END_VAR
VAR
	tCheckingFVP:							TON;//Таймер проеврки ФВН
	tStopTMP:								TON;//Таймер отановки УВП
	tOpenBAV3:								TON;
	iVacuumCameraProcessStage:				INT;//Стадия работывакуумной камеры   
	iCallbackStage:							INT;//Стадия с которой произошел переход в ошибку
	iVacuumCameraLastProcessStage:			INT;//Предыдущая стадия процесса вакуумной камеры
	iVacuumCameraNextProcessStage:			INT;//Следующая стадия процесса вакуумной камеры
	wStatus:								WORD;//Cтатус работы
	xVacuumCameraDevicesAutomode:			BOOL;//Все устрйоства вакуумной камеры в автоматическом режиме
	xLockCommand:							BOOL;//Сигнал о блокировки ввода новой комманды
	xStartFVPCheckinTimerFlag:				BOOL;//Флаг запуска таймера проверки насоса.
	xOpenBAV3timerFlag:						BOOL;
	xStopTMPTimerFlag:						BOOL;
END_VAR

VacuumCameraSetting.tStopTMPtime:=UDINT_TO_TIME((UINT_TO_UDINT(VacuumCameraSetting.uiStopTMPTimeSP)*1000));
VacuumCameraSetting.tOpenBAV3time:=UDINT_TO_TIME((UINT_TO_UDINT(VacuumCameraSetting.uiOpenBAV3TimeSP)*1000));
VacuumCameraSetting.uiStopTMPTimeLeft:=VacuumCameraSetting.uiStopTMPTimeLeft/1000;

tCheckingFVP.IN:=xStartFVPCheckinTimerFlag;
tCheckingFVP.PT:=T#60S;
tCheckingFVP();

tStopTMP.IN:=xStopTMPTimerFlag; 
tStopTMP.PT:=VacuumCameraSetting.tStopTMPtime;
VacuumCameraSetting.tStopTMPTimeLeft:=tStopTMP.ET;
tStopTMP();

tOpenBAV3.IN:=xOpenBAV3timerFlag;
tOpenBAV3.PT:=VacuumCameraSetting.tOpenBAV3time;
tOpenBAV3();


IF ClosedCameraSensore.xValue THEN
	VacuumCamera.xClosed:=TRUE;
ELSE
	VacuumCamera.xClosed:=FALSE;
END_IF

xVacuumCameraDevicesAutomode:=isVacuumCameraDeviceAutoMode;


CASE iVacuumCameraProcessStage OF
	

	VACUUM_CAMERA_PROCESS_STAGE.WAIT:	
	
		IF NOT xLockCommand  THEN
			OperatorCommandHandler();
		ELSE
			CancelOperatorCommand();
		END_IF
		IF xStopAnyProcessCommandFromOperator THEN
			iVacuumCameraNextProcessStage:=VACUUM_CAMERA_PROCESS_STAGE.STOP_ANY_PROCESS;
			xStopAnyProcessCommandFromOperator:=FALSE;
			Status:=VacuumCameraStatusList.STOP_ANY_PROCESS_SIGNAL_FROM_OPERATOR;
		END_IF
		IF NOT isVacuumCameraDeviceAutoMode AND xLockCommand THEN
			Status:=VacuumCameraStatusList.SYSTEM_HAS_ERROR;
			xError:=TRUE;
			wError:=VacuumCameraErrorsList.ALL_DEVICES_DONT_HAVE_AUTOMODE;
		END_IF
		IF xError THEN
			Status:=VacuumCameraStatusList.SYSTEM_HAS_ERROR;
			iVacuumCameraNextProcessStage:=VACUUM_CAMERA_PROCESS_STAGE.ERROR;
		END_IF
		iVacuumCameraProcessStage:=iVacuumCameraNextProcessStage;
		
	
	
	
	VACUUM_CAMERA_PROCESS_STAGE.START_VACUUM_PROCESS:
		iVacuumCameraLastProcessStage:=iVacuumCameraProcessStage;
		iCallBackStage:=iVacuumCameraProcessStage;
		Status:=startVacuumProcess();
		iVacuumCameraProcessStage:=VACUUM_CAMERA_PROCESS_STAGE.WAIT;
		
	VACUUM_CAMERA_PROCESS_STAGE.START_VACUUM_PROCESS_CHECK_FVP_SELECT:
		iVacuumCameraLastProcessStage:=iVacuumCameraProcessStage;
		iCallBackStage:=iVacuumCameraProcessStage;
		Status:=CheckFVPSelect();
		iVacuumCameraProcessStage:=VACUUM_CAMERA_PROCESS_STAGE.WAIT;
		
	VACUUM_CAMERA_PROCESS_STAGE.START_VACUUM_PROCESS_CHECKING_FVP:
		iVacuumCameraLastProcessStage:=iVacuumCameraProcessStage;
		iCallbackStage:=iVacuumCameraProcessStage;
		Status:=CheckingFVP();
		iVacuumCameraProcessStage:=VACUUM_CAMERA_PROCESS_STAGE.WAIT;
		
		
	VACUUM_CAMERA_PROCESS_STAGE.START_VACUUM_PROCESS_FORVACUUMING_PROCESS:
		iVacuumCameraLastProcessStage:=iVacuumCameraProcessStage;
		iCallbackStage:=iVacuumCameraProcessStage;
		Status:=forvacuumingProcess();
		iVacuumCameraProcessStage:=VACUUM_CAMERA_PROCESS_STAGE.WAIT;
		
	VACUUM_CAMERA_PROCESS_STAGE.START_VACUUM_PROCESS_TMP_FORVACUUMING_PROCESS:
		iVacuumCameraLastProcessStage:=iVacuumCameraProcessStage;
		iCallbackStage:=iVacuumCameraProcessStage;
		Status:=forvacuumingWithTMPValve();
		iVacuumCameraProcessStage:=VACUUM_CAMERA_PROCESS_STAGE.WAIT;
		
	VACUUM_CAMERA_PROCESS_STAGE.START_VACUUM_PROCESS_TMP_START:
		iVacuumCameraLastProcessStage:=iVacuumCameraProcessStage;
		iCallbackStage:=iVacuumCameraProcessStage;
		Status:=startTMP();
		iVacuumCameraProcessStage:=VACUUM_CAMERA_PROCESS_STAGE.WAIT;
	
	VACUUM_CAMERA_PROCESS_STAGE.START_VACUUM_PROCESS_COMPLETE_WAIT:
		iVacuumCameraLastProcessStage:=iVacuumCameraProcessStage;
		iCallbackStage:=iVacuumCameraProcessStage;
		Status:=waitVacuumingProcess();
		iVacuumCameraProcessStage:=VACUUM_CAMERA_PROCESS_STAGE.WAIT;
	
	
	VACUUM_CAMERA_PROCESS_STAGE.START_DEVACUUM_PROCESS:
		iVacuumCameraLastProcessStage:=iVacuumCameraProcessStage;
		iCallbackStage:=iVacuumCameraProcessStage;
		Status:=startDevacuumProcess();
		iVacuumCameraProcessStage:=VACUUM_CAMERA_PROCESS_STAGE.WAIT;
		
		
	VACUUM_CAMERA_PROCESS_STAGE.START_DEVACUUM_STOP_TMP:
		iVacuumCameraLastProcessStage:=iVacuumCameraProcessStage;
		iCallbackStage:=iVacuumCameraProcessStage;
		Status:=stopTMP();
		iVacuumCameraProcessStage:=VACUUM_CAMERA_PROCESS_STAGE.WAIT;

		
		
	VACUUM_CAMERA_PROCESS_STAGE.START_DEVACUUM_STOP_FVP:
		iVacuumCameraLastProcessStage:=iVacuumCameraProcessStage;
		iCallbackStage:=iVacuumCameraProcessStage;	
		Status:=stopFVP();
		iVacuumCameraProcessStage:=VACUUM_CAMERA_PROCESS_STAGE.WAIT;
		
	VACUUM_CAMERA_PROCESS_STAGE.START_DEVACUUM_OPEN_CAM:
		iVacuumCameraLastProcessStage:=iVacuumCameraProcessStage;
		iCallbackStage:=iVacuumCameraProcessStage;	
		Status:=devcuumProcessOpenCam();
		iVacuumCameraProcessStage:=VACUUM_CAMERA_PROCESS_STAGE.WAIT;
	
		
	VACUUM_CAMERA_PROCESS_STAGE.STOP_VACUUM_PROCESS:
		iVacuumCameraLastProcessStage:=iVacuumCameraProcessStage;
		iCallbackStage:=iVacuumCameraProcessStage;
		Status:=stopVacuumProcess();
		iVacuumCameraProcessStage:=VACUUM_CAMERA_PROCESS_STAGE.WAIT;
	
	VACUUM_CAMERA_PROCESS_STAGE.STOP_ANY_PROCESS:
		iVacuumCameraLastProcessStage:=iVacuumCameraProcessStage;
		iCallbackStage:=iVacuumCameraProcessStage;
		Status:=operatorStopAnyProcess();
		iVacuumCameraProcessStage:=VACUUM_CAMERA_PROCESS_STAGE.WAIT;
		
		
	VACUUM_CAMERA_PROCESS_STAGE.ERROR:
	
		ErrorHandle();
	
		
END_CASE

VacuumCamera.VacuumCameraProcessStage:=iVacuumCameraProcessStage;

ACTION StartDevacuumProcessCommand:
xStartDevacuumProcessOperatorCommand:=FALSE;
	IF isVacuumCameraDeviceAutoMode THEN
		iVacuumCameraNextProcessStage:=VACUUM_CAMERA_PROCESS_STAGE.START_DEVACUUM_PROCESS;
		xLockCommand:=TRUE;
		wError:=VacuumCameraErrorsList.NO_ERROR;
		RETURN;
	ELSE
		xError:=true;
		wError:=VacuumCameraErrorsList.ALL_DEVICES_DONT_HAVE_AUTOMODE;
		iVacuumCameraNextProcessStage:= VACUUM_CAMERA_PROCESS_STAGE.ERROR;
	END_IF
END_ACTION

ACTION StartVacuumProcessCommand:
	xStartVacuumProcessOperatorCommand:=FALSE;
	IF isVacuumCameraDeviceAutoMode THEN
		iVacuumCameraNextProcessStage:= VACUUM_CAMERA_PROCESS_STAGE.START_VACUUM_PROCESS;
		xLockCommand:=TRUE;
		wError:=VacuumCameraErrorsList.NO_ERROR;
		RETURN;
	END_IF
	IF NOT isVacuumCameraDeviceAutoMode THEN
		xError:=TRUE;
		wError:=VacuumCameraErrorsList.ALL_DEVICES_DONT_HAVE_AUTOMODE;
		iVacuumCameraNextProcessStage:= VACUUM_CAMERA_PROCESS_STAGE.ERROR;
	END_IF
	IF NOT VacuumCamera.xClosed THEN
		xError:=TRUE;
		wError:=VacuumCameraErrorsList.VACUUM_CAMERA_OPEN;
		iVacuumCameraNextProcessStage:= VACUUM_CAMERA_PROCESS_STAGE.ERROR;
	END_IF
END_ACTION

ACTION StopVacuumProcessCommand:
xStartVacuumProcessOperatorCommand:=FALSE;
IF isVacuumCameraDeviceAutoMode THEN
	iVacuumCameraNextProcessStage:=VACUUM_CAMERA_PROCESS_STAGE.STOP_VACUUM_PROCESS;
	xLockCommand:=TRUE;
	TMPBreakingValve.xAutoCommand:=FALSE;
	wError:=VacuumCameraErrorsList.NO_ERROR;
	RETURN;
ELSE
	xError:=TRUE;
	wError:=VacuumCameraErrorsList.ALL_DEVICES_DONT_HAVE_AUTOMODE;
	iVacuumCameraNextProcessStage:= VACUUM_CAMERA_PROCESS_STAGE.ERROR;
	
END_IF
END_ACTION

METHOD PROTECTED CancelOperatorCommand
VAR_INPUT
END_VAR
xStartVacuumProcessOperatorCommand:=FALSE;
xStartDevacuumProcessOperatorCommand:=FALSE;
xStopVacuumProcesOoperatorCommand:=FALSE;
END_METHOD

METHOD PROTECTED CheckFVPSelect : WORD
VAR_INPUT
END_VAR
IF NOT FVP.xStart THEN
			FVP.xAutoCommand:=TRUE;
			CheckFVPSelect:=VacuumCameraStatusList.CHECK_FVP_START_FVP;
END_IF
IF VacuumCamera.xFVPChecked THEN
			iVacuumCameraNextProcessStage:=VACUUM_CAMERA_PROCESS_STAGE.START_VACUUM_PROCESS_FORVACUUMING_PROCESS;
			CheckFVPSelect:=VacuumCameraStatusList.FVP_CHECK_COMPLETED;
ELSE
			iVacuumCameraNextProcessStage:=VACUUM_CAMERA_PROCESS_STAGE.START_VACUUM_PROCESS_CHECKING_FVP;
			xStartFVPCheckinTimerFlag:=TRUE;
END_IF
END_METHOD

METHOD PROTECTED CheckingFVP : WORD
VAR_INPUT
END_VAR
CheckingFVP:=VacuumCameraStatusList.CHECK_FVP_START_TIMER;		
IF tCheckingFVP.Q THEN
			IF FVPPressure.rPressure <= VacuumCameraSetting.rForvacPresureToCheckFVP THEN
				CheckingFVP:=VacuumCameraStatusList.CHECK_FVP_COMPLETE;
				VacuumCamera.xFVPChecked:=TRUE;
				iVacuumCameraNextProcessStage:=VACUUM_CAMERA_PROCESS_STAGE.START_VACUUM_PROCESS_FORVACUUMING_PROCESS;
			ELSE
				CheckingFVP:=VacuumCameraStatusList.CHECK_FVP_FAILED;
				iVacuumCameraNextProcessStage:=VACUUM_CAMERA_PROCESS_STAGE.ERROR;
				wError:=VacuumCameraErrorsList.FVP_CHECK_FAIL;
				xError:=TRUE;
			END_IF
	xStartFVPCheckinTimerFlag:=FALSE;
END_IF
END_METHOD

METHOD PROTECTED CloseAllvalves
VAR_INPUT
END_VAR
IF BAV1.xOpened THEN
	BAV1.xAutoCommand:=FALSE;
END_IF
IF BAV2.xOpened THEN
	BAV2.xAutoCommand:=FALSE;
END_IF
IF BAV3.xOpened THEN
	BAV3.xAutoCommand:=FALSE;
END_IF
IF TMPBreakingValve.xOpened THEN
	TMPBreakingValve.xAutoCommand:=FALSE;
END_IF
END_METHOD

METHOD PROTECTED devcuumProcessOpenCam : WORD
VAR_INPUT
END_VAR
IF BAV3.xClosed THEN
	BAV3.xAutoCommand:=TRUE;
	xOpenBAV3timerFlag:= TRUE;
	devcuumProcessOpenCam:=VacuumCameraStatusList.BAV3OPENED;
END_IF
IF tOpenBAV3.Q THEN
	xOpenBAV3timerFlag:=FALSE;
	BAV3.xAutoCommand:=FALSE;
	xLockCommand:=FALSE;
	devcuumProcessOpenCam:=VacuumCameraStatusList.STOP_SYSTEM_COMPLITE;
	iVacuumCameraNextProcessStage:= VACUUM_CAMERA_PROCESS_STAGE.WAIT;
END_IF
END_METHOD

METHOD PRIVATE ErrorHandle : WORD
VAR_INPUT
END_VAR
IF xProcessResumeCommand THEN
	xProcessResumeCommand:=FALSE;
	iVacuumCameraNextProcessStage:=iCallbackStage;
	iVacuumCameraProcessStage:=VACUUM_CAMERA_PROCESS_STAGE.WAIT;
	xError:=FALSE;
	wError:=VacuumCameraErrorsList.NO_ERROR;
END_IF
IF xProcessAbort THEN
	xProcessAbort:=FALSE;
	iVacuumCameraNextProcessStage:=VACUUM_CAMERA_PROCESS_STAGE.WAIT;
	iVacuumCameraProcessStage:=VACUUM_CAMERA_PROCESS_STAGE.WAIT;
	xError:=FALSE;
	xLockCommand:=FALSE;
	wError:=VacuumCameraErrorsList.NO_ERROR;
	Status:=VacuumCameraStatusList.SYSTEM_READY_AND_WAIT_COMMAND;
END_IF
END_METHOD

METHOD PROTECTED forvacuumingProcess : WORD
VAR_INPUT
	
END_VAR
IF BAV1.xOpened THEN
	forvacuumingProcess:=VacuumCameraStatusList.START_FORVAC_PROCESS;
	IF CameraPressure.rPressure < 15 THEN
		iVacuumCameraNextProcessStage:= VACUUM_CAMERA_PROCESS_STAGE.START_VACUUM_PROCESS_TMP_FORVACUUMING_PROCESS;
		forvacuumingProcess:=VacuumCameraStatusList.FORVAC_COMPLETE;
	END_IF
ELSE
	BAV1.xAutoCommand:=TRUE;
END_IF
END_METHOD

METHOD PROTECTED forvacuumingWithTMPValve : WORD
VAR_INPUT
END_VAR
IF BAV2.xClosed THEN
	BAV2.xAutoCommand:=TRUE;
END_IF
forvacuumingWithTMPValve:=VacuumCameraStatusList.FORVAC_WITH_TMP_VALVE;
IF BAV1.xOpened AND BAV2.xOpened AND CameraPressure.rPressure<VacuumCameraSetting.rPressureToStartTMPSP THEN
	iVacuumCameraNextProcessStage:= VACUUM_CAMERA_PROCESS_STAGE.START_VACUUM_PROCESS_TMP_START;
	forvacuumingWithTMPValve:=VacuumCameraStatusList.FORVAC_WITH_TMP_VALVE_COMPLETE;
END_IF
END_METHOD

METHOD PROTECTED OperatorCommandHandler
VAR_INPUT
END_VAR
IF xStartVacuumProcessOperatorCommand THEN
	StartVacuumProcessCommand();
END_IF

IF xStartDevacuumProcessOperatorCommand THEN
	StartDevacuumProcessCommand();
END_IF

IF xStopVacuumProcesOoperatorCommand THEN
	StopVacuumProcessCommand();
END_IF

wStatus:=VacuumCameraStatusList.SYSTEM_READY_AND_WAIT_COMMAND;
END_METHOD

METHOD PROTECTED operatorStopAnyProcess : WORD
VAR_INPUT
END_VAR
xLockCommand:=FALSE;
xOpenBAV3timerFlag:=FALSE;
xStartFVPCheckinTimerFlag:=FALSE;
xStopTMPTimerFlag:=FALSE;
operatorStopAnyProcess:=VacuumCameraStatusList.OPERATOR_STOPED_PROCESS_COMPLETE;
iVacuumCameraNextProcessStage:= VACUUM_CAMERA_PROCESS_STAGE.WAIT;
END_METHOD

METHOD PROTECTED startDevacuumProcess : WORD
VAR_INPUT
END_VAR

		TMP.xAutoCommand:=FALSE;
		TMPBreakingValve.xAutoCommand:=TRUE;
		xStopTMPTimerFlag:=TRUE;
		iVacuumCameraNextProcessStage:= VACUUM_CAMERA_PROCESS_STAGE.START_DEVACUUM_STOP_TMP;
		startDevacuumProcess:=VacuumCameraStatusList.STOP_TMP_PROCESS;
(*ELSIF BAV2.xClosed AND TMP.xPumpNotOperating THEN
		FVP.xAutoCommand:=FALSE;
		iVacuumCameraNextProcessStage:= VACUUM_CAMERA_PROCESS_STAGE.START_DEVACUUM_STOP_FVP;
		startDevacuumProcess:=VacuumCameraStatusList.STOP_FVP_PROCESS;
END_IF*)
END_METHOD

METHOD PROTECTED startTMP : WORD
VAR_INPUT
END_VAR
		startTMP:=VacuumCameraStatusList.TMP_IS_STARTED;
		IF BAV1.xOpened THEN
			BAV1.xAutoCommand:=FALSE;
		END_IF
		IF BAV1.xClosed AND NOT TMP.xStart THEN
			TMP.xAutoCommand:=TRUE;
			startTMP:=VacuumCameraStatusList.TMP_IS_STARTED;
		END_IF
		IF TMP.xNormalOperation THEN
			startTMP:=VacuumCameraStatusList.TMP_IS_RUN;
			iVacuumCameraNextProcessStage:=VACUUM_CAMERA_PROCESS_STAGE.START_VACUUM_PROCESS_COMPLETE_WAIT;
		END_IF
		IF TMP.xError THEN
			TMP.xAutoCommand:=FALSE;
			xError:=TRUE;
			wError:=VacuumCameraErrorsList.TMP_ERROR_FROM_START;
			iVacuumCameraProcessStage:=VACUUM_CAMERA_PROCESS_STAGE.ERROR;
			return;
		END_IF
END_METHOD

METHOD PROTECTED startVacuumProcess : WORD
VAR_INPUT
END_VAR
IF isVacuumCameraDeviceAutoMode AND isVacuumCameraClosed THEN
			IF isAllValvesClosed THEN
				iVacuumCameraNextProcessStage:=VACUUM_CAMERA_PROCESS_STAGE.START_VACUUM_PROCESS_CHECK_FVP_SELECT;
				startVacuumProcess:=VacuumCameraStatusList.START_VACUUM_PROCESS;
			ELSE
				CloseAllvalves();
			END_IF
		ELSE
			wError:= VacuumCameraErrorsList.ALL_DEVICES_DONT_HAVE_AUTOMODE;
			xError:=TRUE;
			startVacuumProcess:=VacuumCameraStatusList.SYSTEM_HAS_ERROR;
			iVacuumCameraNextProcessStage:=VACUUM_CAMERA_PROCESS_STAGE.ERROR;
		END_IF
END_METHOD

METHOD PRIVATE stopFVP : WORD
VAR_INPUT
END_VAR
IF BAV1.xOpened THEN
	BAV1.xAutoCommand:=FALSE;
END_IF

		

	
	
	VacuumCamera.xCameraIsVaccumed:=FALSE;
	FVP.xAutoCommand:=FALSE;
	//xLockCommand:=FALSE;
	stopFVP:=VacuumCameraStatusList.STOP_FVP_PROCESS_DONE;
	iVacuumCameraNextProcessStage:=VACUUM_CAMERA_PROCESS_STAGE.START_DEVACUUM_OPEN_CAM;
END_METHOD

METHOD stopTMP : WORD
VAR_INPUT
END_VAR
stopTMP:=VacuumCameraStatusList.STOP_TMP_PROCESS;

IF tStopTMP.Q THEN
		TMPBreakingValve.xAutoCommand:=FALSE;
		VacuumCamera.xCameraIsVaccumed:=FALSE;
		BAV2.xAutoCommand:=FALSE;
		xStopTMPTimerFlag:=FALSE;
		iVacuumCameraNextProcessStage:=VACUUM_CAMERA_PROCESS_STAGE.START_DEVACUUM_STOP_FVP;
		stopTMP:=VacuumCameraStatusList.STOP_TMP_DONE;
		
END_IF
END_METHOD

METHOD PRIVATE stopVacuumProcess : WORD
VAR_INPUT
END_VAR
		stopVacuumProcess:=VacuumCameraStatusList.STOP_TMP_PROCESS;
		IF BAV1.xOpened THEN
			BAV1.xAutoCommand:=FALSE;
		END_IF	

		IF TMP.xStart THEN
			TMP.xAutoCommand:=FALSE;
		END_IF
		IF NOT TMP.xAutoCommand THEN
			//TMPBreakingValve.xAutoCommand:=TRUE;
			xStopTMPTimerFlag:=TRUE;
		END_IF
	
		
		IF tStopTMP.Q THEN
			TMPBreakingValve.xAutoCommand:=FALSE;
			Vacuumcamera.xCameraIsVaccumed:=FALSE;
			VacuumCamera.xFVPChecked:=FALSE;
			xStopTMPTimerFlag:=FALSE;
			BAV2.xAutoCommand:=FALSE;
			FVP.xAutoCOmmand:=FALSE;
			xLockCommand:=FALSE;
			stopVacuumProcess:=VacuumCameraStatusList.STOP_SYSTEM_COMPLITE;
			iVacuumCameraNextProcessStage:=VACUUM_CAMERA_PROCESS_STAGE.WAIT;
		END_IF
END_METHOD

METHOD waitVacuumingProcess : WORD
VAR_INPUT
END_VAR
waitVacuumingProcess:=VacuumCameraStatusList.CAMERA_IS_VACUUMING;
IF CameraPressure.rPressure<VacuumCameraSetting.rPressureProcessComplete THEN
			VacuumCamera.xCameraIsVaccumed:=TRUE;
			xLockCommand:=FALSE;
			iVacuumCameraNextProcessStage:=VACUUM_CAMERA_PROCESS_STAGE.WAIT;
			waitVacuumingProcess:=VacuumCameraStatusList.VACUUM_DONE;
END_IF
END_METHOD

PROPERTY PROTECTED isAllValvesClosed : BOOL
GET
isAllValvesClosed:=BAV1.xClosed AND BAV2.xClosed AND BAV3.xClosed AND NOT TMPBreakingValve.xOpened;
END_GET
END_PROPERTY

PROPERTY PROTECTED isFVPChecked : BOOL
GET
isFVPChecked:=Vacuumcamera.xFVPChecked;
END_GET
SET
VacuumCamera.xFVPChecked:=isFVPChecked;
END_SET
END_PROPERTY

PROPERTY isOperatorCommandEntryLocked : BOOL
GET
isOperatorCommandEntryLocked:=THIS^.xLockCommand;
END_GET
END_PROPERTY

PROPERTY PROTECTED isVacuumCameraClosed : BOOL
GET
isVacuumCameraClosed:=VacuumCamera.xClosed;
END_GET
END_PROPERTY

PROPERTY PRIVATE isVacuumCameraDeviceAutoMode : BOOL
GET
IF  BAV1Setting.xAutoMode AND BAV2Setting.xAutoMode AND BAV3Setting.xAutoMode AND TMPSetting.xAutoMode AND FVPSetting.xAutoMode AND TMPBreakingValveSetting.xAutoMode  THEN
	isVacuumCameraDeviceAutoMode:=TRUE;
ELSE
	isVacuumCameraDeviceAutoMode:=FALSE;
END_IF
END_GET
END_PROPERTY

END_FUNCTION_BLOCK

// Function Blocks/VacuumCamera/Pumping/VacuumingCameraWithSHV
FUNCTION_BLOCK VacuumingCameraWithSHV
VAR_INPUT
	//PreInit:		itfPreAction;
	refVacuumCamera: 	REFERENCE TO udtVacuumCamera;
	refVacuumProccess: 	REFERENCE TO udtVacuumProcess;
	refState:			REFERENCE TO udtVacuumProcessState;
	StartUnitSetting: 	udtStartUnitProcessSetting;
	Devacuumsetting:	udtDevacuumUnitProcessSetting;
	RevacuumSetting:	udtRevacuumProcessSetting;
	refBAV1Small:		REFERENCE TO udtValve;
	refBAV1Big:			REFERENCE TO udtValve;
	BAV1AutoMode:		BOOL;
	refBAV2:			REFERENCE TO udtValve;
	BAV2AutoMode:		BOOL;
	refBAV3Small:		REFERENCE TO udtValve;
	refBAV3Big:			REFERENCE TO udtValve;
	BAV3SmallAuto:		BOOL;
	BAV3BigAuto:		BOOL;
	refSHV:				REFERENCE TO udtValve;
	SHVAutoMode:		BOOL;
	refFVP:				REFERENCE TO udtFVP;
	FVPAutoMode:		BOOL;
	refTMP:				REFERENCE TO udtTMPDigital;
	refTMPSetting: 		REFERENCE TO udtTMPDigitalSetting;
	refFVPPressure:		REFERENCE TO udtPressureSensore;
	refCameraPressure:	REFERENCE TO udtPressureSensore;
END_VAR
VAR_OUTPUT
	xError:			BOOL;
	wStatus:		WORD;
END_VAR
VAR
	StartUnitProcessStage:				INT;
	DevacuumProcessStage:				INT;
	RevacuumProcessStage:				INT;
	StopUnitProcessStage:				INT;
	
	StartUnitFVPCheckTimer:				TON;
	DevacuumWaitTimer:					TON;
	RevacuumWaitTimer:					TON;
	
	Init: 								BOOL;
	StartUnitProcessStartFVpCheckTimer:	BOOL;
	StartDevacummWaitTimer:				BOOL;
	StartRevacuumWaitTimer:				BOOL;
	
	StartUnitProcessComplete: 			BOOL; //Процесс запуска вакуумного оборудования успешно завершен
	StarUnitProcessError:				BOOL; //Ошибка запуска оборудования
	
	DevacuumProcessComplete:			BOOL;
	DevacuumProcessError:				BOOL;
	
	RevacuumProcessComplete:			BOOL;
	RevacuumProcessError:				BOOL;
	
	StopUnitProcessComplete:			BOOL;
	StopUnitProcessError:				BOOL;
	_xCommandLock:						BOOL;//Блокировка комманд
	_iNextStage:						INT;//Следующая стадия
	_iCallbackStage:					INT;//Стадия возвращения при обработки ошибки
	_iLastStage:						INT;//Последняя отрабтанная стадия
	
	
END_VAR

IF NOT Init THEN
	//PreInit.PreAction();
	StartUnitFVPCheckTimer.IN:=StartUnitProcessStartFVpCheckTimer;
	DevacuumWaitTimer.IN:=StartDevacummWaitTimer;
	RevacuumWaitTImer.IN:=StartRevacuumWaitTimer;
	Init:=TRUE;
END_IF;


refVacuumProccess.Status.bStatus.BAV1NotAutoMode:=	NOT BAV1AutoMode;
refVacuumProccess.Status.bStatus.BAV2NotAutoMode:=	NOT BAV2autoMode;
refVacuumProccess.Status.bStatus.BAV3SmallNotAutoMode:=	NOT BAV3SmallAuto;
refVacuumProccess.Status.bStatus.BAV3BigNotAutoMode:= NOT BAV3BigAuto;
refVacuumProccess.Status.bStatus.FVPNotAutoMode:=	NOT FVPAutoMode;
refVacuumProccess.Status.bStatus.FVPNotPowerOn:=	NOT refFVP.xPowerOnFeedBack;
refVacuumProccess.Status.bStatus.SHVNotAutoMode:=	NOT SHVAutoMode;
refVacuumProccess.Status.bStatus.TMPNotAutoMode:=	NOT refTMPSetting.xAutoMode;
refVacuumProccess.Status.bStatus.TMPNotPowerOn:=	NOT refTMP.xPowerOnFeedBack;
refVacuumProccess.Status.bStatus.StartStatusProcessError:=THIS^.StarUnitProcessError;

StartUnitFVPCheckTimer(PT:=StartUnitSetting.FVPCheckTime);
DevacuumWaitTimer(PT:=Devacuumsetting.WaitTime);
RevacuumWaitTimer(PT:=RevacuumSetting.WaitTime);

CASE refVacuumProccess.Stage OF
	VacuumStage.WAIT:
		THIS^._commandHandler();
		THIS^.refVacuumProccess.Stage:=THIS^._iNextStage;
	
		 {region "old"}
		(*IF refVacuumProccess.xStartUnit AND refVacuumProccess.Status.Status=0 THEN
			refVacuumProccess.xStartUnit:=FALSE;
			refVacuumProccess.Stage:=VacuumStage.START_UNIT;
		ELSIF refVacuumProccess.xStartUnit AND refVacuumProccess.Status.Status <> 0 THEN
			refVacuumProccess.xStartUnit := FALSE;
			refVacuumProccess.Stage:=VacuumStage.ERROR;
		END_IF
		IF refVacuumProccess.xStartDevacuumProcess AND refVacuumProccess.Status.Status=0 THEN
			refVacuumProccess.xStartDevacuumProcess:=FALSE;
			refVacuumProccess.Stage:=VacuumStage.DEVACUUM;
		ELSIF refVacuumProccess.xStartDevacuumProcess AND refVacuumProccess.Status.Status <> 0 THEN
			refVacuumProccess.xStartDevacuumProcess := FALSE;
			refVacuumProccess.Stage:=VacuumStage.ERROR;
		END_IF
		IF refVacuumProccess.xStartRevacuumProccess AND refVacuumProccess.Status.Status=0 AND refState.UnitTurnOn THEN
			refVacuumProccess.xStartRevacuumProccess:=FALSE;
			refVacuumProccess.Stage:=VacuumStage.REVACUUM;
		ELSE
			refVacuumProccess.xStartRevacuumProccess := FALSE;
			refVacuumProccess.Stage:=VacuumStage.ERROR;
		END_IF
		IF refVacuumProccess.xStopUnit AND refVacuumProccess.Status.Status=0 THEN
			refVacuumProccess.xStopUnit:=FALSE;
			refVacuumProccess.Stage:=VacuumStage.STOP_UNIT;
		ELSE
			refVacuumProccess.xStopUnit := FALSE;
			refVacuumProccess.Stage:=VacuumStage.ERROR;
		END_IF*)
		{end_region}
		
	VacuumStage.START_UNIT:
		THIS^._iCallbackStage:=THIS^.refVacuumProccess.Stage;
		StartUnit();
		IF StartUnitProcessComplete AND NOT StarUnitProcessError THEN
			THIS^._iNextStage:=VacuumStage.START_UNIT_COMPETE;
			 refVacuumProccess.Stage:=VacuumStage.WAIT;
		ELSIF StarUnitProcessError THEN
			refVacuumProccess.Stage:=VacuumStage.ERROR;
		END_IF
		
	VacuumStage.START_UNIT_COMPETE:
		THIS^._iCallbackStage:=THIS^.refVacuumProccess.Stage;
		THIS^.refState.UnitTurnOn:=TRUE;
		THIS^.refState.VacuumedUnit:=TRUE;
		THIS^.refState.DevacuumedUnit:=FALSE;
		THIS^.refState.UnitTurnOff:=FALSE;
		THIS^._iNextStage:=VacuumStage.WAIT;
		refVacuumProccess.Stage:=VacuumStage.WAIT;
	
	VacuumStage.DEVACUUM:
		THIS^._iCallbackStage:=THIS^.refVacuumProccess.Stage;
		Devacuum();
		IF DevacuumProcessComplete THEN
			THIS^._iNextStage:=VacuumStage.DEVACUUM_COMPLETE;
			 refVacuumProccess.Stage:=VacuumStage.WAIT;
		ELSIF DevacuumProcessError THEN
			refVacuumProccess.Stage:=VacuumStage.ERROR;
		END_IF
	
	VacuumStage.DEVACUUM_COMPLETE:
		THIS^._iCallbackStage:=THIS^.refVacuumProccess.Stage;
		THIS^.refState.DevacuumedUnit:=TRUE;
		THIS^.refState.VacuumedUnit:=FALSE;
		THIS^._iNextStage:=VacuumStage.WAIT;
		refVacuumProccess.Stage:=VacuumStage.WAIT;
	
	VacuumStage.REVACUUM:
		THIS^._iCallbackStage:=THIS^.refVacuumProccess.Stage;
		Revacuum();
		IF RevacuumProcessComplete THEN
			THIS^._iNextStage:=VacuumStage.REVACUUM_COMPLETE;
			refVacuumProccess.Stage:=VacuumStage.WAIT;
		ELSIF RevacuumProcessError THEN
			refVacuumProccess.Stage:=VacuumStage.ERROR;
		END_IF
	VacuumStage.REVACUUM_COMPLETE:
		THIS^._iCallbackStage:=THIS^.refVacuumProccess.Stage;
		THIS^.refState.DevacuumedUnit:=FALSE;
		THIS^.refState.VacuumedUnit:=TRUE;
		THIS^._iNextStage:=VacuumStage.WAIT;
		refVacuumProccess.Stage:=VacuumStage.WAIT;
	
	VacuumStage.STOP_UNIT:
		THIS^._iCallbackStage:=THIS^.refVacuumProccess.Stage;
		StopUnit();
		IF StopUnitProcessComplete THEN
			THIS^._iNextStage:=VacuumStage.STOP_UNIT_COMPLETE;
			refVacuumProccess.Stage:=VacuumStage.WAIT;
		ELSIF StopUnitProcessError THEN
			refVacuumProccess.Stage:=VacuumStage.ERROR;
		END_IF
	VacuumStage.STOP_UNIT_COMPLETE:
		THIS^._iCallbackStage:=THIS^.refVacuumProccess.Stage;
		THIS^.refState.DevacuumedUnit:=FALSE;
		THIS^.refState.VacuumedUnit:=FALSE;
		THIS^.refState.UnitTurnOn:=FALSE;
		THIS^.refState.UnitTurnOff:=TRUE;
		THIS^._iNextStage:=VacuumStage.WAIT;	 
		refVacuumProccess.Stage:=VacuumStage.WAIT;
		
	VacuumStage.ERROR:
		IF RevacuumProcessError THEN
			RevacuumProcessStage:=RevacuumStage.WAIT;
		END_IF
		IF StopUnitProcessError THEN
			StopUnitProcessStage:= StopUnitStage.WAIT;
		END_IF
		
	//TODO: Сделать что-нибудь
		IF refVacuumProccess.ResetError THEN
			RevacuumProcessError:=FALSE;
			refVacuumProccess.Stage:=VacuumStage.WAIT;
		END_IF
END_CASE

ACTION CloseAllValves:
THIS^.refBAV3Big.xAutoCommand:=FALSE;
THIS^.refBAV3Small.xAutoCommand:=FALSE;
THIS^.refBAV1Big.xAutoCommand:=FALSE;
THIS^.refBAV1Small.xAutoCommand:=FALSE;
THIS^.refBAV2.xAutoCommand:=FALSE;
THIS^.refSHV.xAutoCommand:=FALSE;
END_ACTION

METHOD PUBLIC Devacuum : WORD
VAR_INPUT
END_VAR
CASE THIS^.DevacuumProcessStage OF
	DevacuumUnitStage.WAIT:
		THIS^.DevacuumProcessStage:=DevacuumUnitStage.CHECK_SYSTEM;
	DevacuumUnitStage.CHECK_SYSTEM:
		IF THIS^.refBAV3Big.xOpened OR THIS^.refBAV3Small.xOpened THEN
			THIS^.DevacuumProcessStage:=DevacuumUnitStage.COMPLETE;
		ELSE
			THIS^.DevacuumProcessStage:=DevacuumUnitStage.CLOSE_VALVES;
		END_IF
	DevacuumUnitStage.CLOSE_VALVES:
		IF THIS^.refBAV1Big.xOpened THEN
			THIS^.refBAV1Big.xAutoCommand:=FALSE;
		END_IF
		IF THIS^.refBAV1Small.xOpened THEN
			THIS^.refBAV1Small.xAutoCommand:=FALSE;
		END_IF
		IF THIS^.refSHV.xOpened THEN
			THIS^.refSHV.xAutoCommand:=FALSE;
		END_IF
		IF 	THIS^.refBAV1Big.xClosed AND
			THIS^.refBAV1Small.xClosed AND
			THIS^.refSHV.xClosed THEN
			THIS^.StartDevacummWaitTimer:=TRUE;
			THIS^.DevacuumProcessStage:=DevacuumUnitStage.WAIT_TIME;
		END_IF
	//Закрытие всех клапанов кроме BAV2
	DevacuumUnitStage.WAIT_TIME:
		IF THIS^.DevacuumWaitTimer.Q THEN
			THIS^.StartDevacummWaitTimer:=FALSE;
			THIS^.DevacuumProcessStage:=DevacuumUnitStage.OPEN_VALVE;
		END_IF
	DevacuumUnitStage.OPEN_VALVE:
		IF THIS^.refBAV3Small.xClosed THEN
			THIS^.refBAV3Small.xAutoCommand:=TRUE;
		END_IF
		IF THIS^.refBAV3Big.xClosed THEN
			THIS^.refBAV3Big.xAutoCommand:=TRUE;
		END_IF
		IF THIS^.refBAV3Small.xOpened AND THIS^.refBAV3Big.xOpened THEN
			THIS^.DevacuumProcessStage:=DevacuumUnitStage.COMPLETE;
		END_IF
	//Открытие клапана напуска
	DevacuumUnitStage.COMPLETE:
		THIS^.DevacuumProcessComplete:=TRUE;
		THIS^.DevacuumProcessStage:=DevacuumUnitStage.WAIT;
	DevacuumUnitStage.ERROR:
END_CASE
END_METHOD

METHOD Revacuum : WORD
VAR_INPUT
END_VAR
CASE THIS^.RevacuumProcessStage OF
	RevacuumStage.WAIT:
		THIS^.refVacuumProccess.xStartRevacuumProccess:=FALSE;
		THIS^.RevacuumProcessStage:=RevacuumStage.CLOSE_BAV3;
	RevacuumStage.CLOSE_BAV3:
		IF THIS^.refBAV3Big.xOpened THEN
			THIS^.refBAV3Big.xAutoCommand:=FALSE;
		END_IF
		IF THIS^.refBAV3Small.xOpened THEN
			THIS^.refBAV3Small.xAutoCommand:=FALSE;
		END_IF
		IF THIS^.refBAV3Small.xError OR THIS^.refBAV3Big.xError THEN
			THIS^.RevacuumProcessStage:=RevacuumStage.ERROR;
		END_IF
		IF THIS^.refBAV3Big.xClosed AND THIS^.refBAV3Small.xClosed THEN
			THIS^.RevacuumProcessStage:=RevacuumStage.CLOSE_TMP_VALVE;
		END_IF
	RevacuumStage.CLOSE_TMP_VALVE:
		IF THIS^.refBAV2.xOpened THEN
			THIS^.refBAV2.xAutoCommand:=FALSE;
		END_IF
		IF THIS^.refBAV2.xClosed THEN
			THIS^.StartRevacuumWaitTimer:=TRUE;
			THIS^.RevacuumProcessStage:=RevacuumStage.WAIT_TIMER;
		END_IF
	RevacuumStage.WAIT_TIMER:
		IF THIS^.RevacuumWaitTimer.Q THEN
			IF THIS^.refBAV3Small.xClosed AND THIS^.refBAV3Big.xClosed AND THIS^.refBAV2.xClosed THEN
				THIS^.StartRevacuumWaitTimer:=FALSE;
				THIS^.RevacuumProcessStage:=RevacuumStage.ERROR;
			ELSE
				THIS^.StartRevacuumWaitTimer:=FALSE;
				THIS^.RevacuumProcessStage:=RevacuumStage.ERROR;
			END_IF
		END_IF
	RevacuumStage.OPEN_BAV1SMALL:
		ValveOpen(	Valve:=THIS^.refBAV1Small,
				 	Stage:=THIS^.RevacuumProcessStage,
				 	Pressure:=THIS^.StartUnitSetting.CamPressureForBAV1LargeOpen,
					NextStage:=RevacuumStage.OPEN_BAV1BIG,
					ErrorStage:=RevacuumStage.ERROR);
	RevacuumStage.OPEN_BAV1BIG:
		ValveOpen(	Valve:=THIS^.refBAV1Big,
				 	Stage:=THIS^.RevacuumProcessStage,
				 	Pressure:=THIS^.refTMPSetting.rMinimalCameraPressure,
					NextStage:=RevacuumStage.OPEN_BAV2,
					ErrorStage:=RevacuumStage.ERROR);
	RevacuumStage.OPEN_BAV2:
		ValveOpen(	Valve:=THIS^.refBAV2,
				 	Stage:=THIS^.RevacuumProcessStage,
				 	Pressure:=THIS^.refTMPSetting.rMinimalCameraPressure,
					NextStage:=RevacuumStage.OPEN_SHV,
					ErrorStage:=RevacuumStage.ERROR);
	RevacuumStage.OPEN_SHV:
		IF THIS^.refBAV1Big.xOpened THEN
			THIS^.refBAV1Big.xAutoCommand:=FALSE;
		END_IF
		IF THIS^.refBAV1Small.xOpened THEN
			THIS^.refBAV1Small.xAutoCommand:=FALSE;
		END_IF
		IF 	THIS^.refBAV1Big.xClosed AND 
			THIS^.refBAV1Small.xClosed AND 
			(THIS^.refCameraPressure.rPressure<=THIS^.refTMPSetting.rMinimalCameraPressure) THEN
			THIS^.refSHV.xAutoCommand:=TRUE;
		END_IF
		IF THIS^.refSHV.xOpened THEN
			THIS^.RevacuumProcessStage:= RevacuumStage.COMPLETE;
		END_IF
	RevacuumStage.COMPLETE:
		IF THIS^.refCameraPressure.rPressure <=THIS^.StartUnitSetting.StartUntiFinallyPressure THEN
			THIS^.RevacuumProcessStage:=RevacuumStage.WAIT;
			THIS^.RevacuumProcessComplete:=TRUE;
		END_IF
	RevacuumStage.ERROR:
		THIS^.RevacuumProcessError:=TRUE;
		
END_CASE
END_METHOD

METHOD PUBLIC StartUnit : WORD
VAR_INPUT
END_VAR
VAR
	
END_VAR
CASE THIS^.StartUnitProcessStage OF
	StartUnitStage.WAIT:
		THIS^.StartUnitProcessStage:=StartUnitStage.CLOSE_VALVES;
	StartUnitStage.CLOSE_VALVES:
		CloseAllValves();
		IF THIS^.isAllvalveClosed THEN
			THIS^.StartUnitProcessStage:=StartUnitStage.START_FVP;
		END_IF
		
	StartUnitStage.START_FVP:
		THIS^.refFVP.xAutoCommand:=TRUE;
		IF THIS^.refFVP.xTurnOn THEN
			THIS^.StartUnitProcessStartFVpCheckTimer:=TRUE;
			THIS^.StartUnitProcessStage:=StartUnitStage.CHECK_FVP;
		END_IF
	StartUnitStage.CHECK_FVP:
		IF THIS^.StartUnitFVPCheckTimer.Q AND THIS^.refCameraPressure.rPressure <= THIS^.StartUnitSetting.FVPCheckPressure THEN
			THIS^.StartUnitProcessStartFVpCheckTimer:=FALSE;
			THIS^.StartUnitProcessStage:=StartUnitStage.OPEN_FORVACUUM_LINE_VALVE_SMALL;
		ELSIF THIS^.StartUnitFVPCheckTimer.Q AND NOT (THIS^.refCameraPressure.rPressure <= THIS^.StartUnitSetting.FVPCheckPressure) THEN
			THIS^.StartUnitProcessStartFVpCheckTimer:=FALSE;
			THIS^.StartUnitProcessStage:=StartUnitStage.ERROR;
		END_IF
	StartUnitStage.OPEN_FORVACUUM_LINE_VALVE_SMALL:
		ValveOpen(	Valve:=THIS^.refBAV1Small,
				 	Stage:=THIS^.StartUnitProcessStage,
				 	Pressure:=THIS^.StartUnitSetting.CamPressureForBAV1LargeOpen,
					NextStage:=StartUnitStage.OPEN_FORVACUUM_LINE_VALVE_LARGE,
					ErrorStage:=StartUnitStage.ERROR);

	StartUnitStage.OPEN_FORVACUUM_LINE_VALVE_LARGE:
		ValveOpen(	Valve:=THIS^.refBAV1Big,
				 	Stage:=THIS^.StartUnitProcessStage,
				 	Pressure:=THIS^.refTMPSetting.rMinimalCameraPressure,
					NextStage:=StartUnitStage.OPEN_TMP_VALVE,
					ErrorStage:=StartUnitStage.ERROR);

	StartUnitStage.OPEN_TMP_VALVE:
		ValveOpen(	Valve:=THIS^.refBAV2,
				 	Stage:=THIS^.StartUnitProcessStage,
				 	Pressure:=THIS^.refTMPSetting.rMinimalCameraPressure,
					NextStage:=StartUnitStage.START_TMP,
					ErrorStage:=StartUnitStage.ERROR);
	StartUnitStage.START_TMP:
		IF 	(THIS^.refCameraPressure.rPressure <= THIS^.refTMPSetting.rMinimalCameraPressure) 
		AND (THIS^.refFVPPressure.rPressure<=THIS^.refTMPSetting.rMinimalForvaccumLinePressure) THEN
			THIS^.refTMP.xAutoCommand:=TRUE;
		END_IF
		IF THIS^.refTMP.xNormalOperation THEN
			THIS^.StartUnitProcessStage:= StartUnitStage.OPEN_SHV;
		END_IF
	StartUnitStage.OPEN_SHV:
		IF THIS^.refBAV1Big.xOpened THEN
			THIS^.refBAV1Big.xAutoCommand:=FALSE;
		END_IF
		IF THIS^.refBAV1Small.xOpened THEN
			THIS^.refBAV1Small.xAutoCommand:=FALSE;
		END_IF
		IF 	THIS^.refBAV1Big.xClosed AND 
			THIS^.refBAV1Small.xClosed AND 
			(THIS^.refCameraPressure.rPressure<=THIS^.refTMPSetting.rMinimalCameraPressure) THEN
			THIS^.refSHV.xAutoCommand:=TRUE;
		END_IF
		IF THIS^.refSHV.xOpened THEN
			THIS^.StartUnitProcessStage:= StartUnitStage.COMPLETE;
		END_IF
	StartUnitStage.COMPLETE:
		IF THIS^.refCameraPressure.rPressure <=THIS^.StartUnitSetting.StartUntiFinallyPressure THEN
			THIS^.StartUnitProcessStage:=StartUnitStage.WAIT;
			THIS^.StartUnitProcessComplete:=TRUE;
		END_IF
	StartUnitStage.ERROR:
		THIS^.refTMP.xAutoCommand:=FALSE;
		THIS^.refFVP.xAutoCommand:=FALSE;
		CloseAllValves();
		THIS^.StarUnitProcessError:=TRUE;
		
END_CASE
END_METHOD

METHOD PUBLIC StopUnit : WORD
VAR_INPUT
END_VAR
CASE THIS^.StopUnitProcessStage OF
	StopUnitStage.WAIT:
		THIS^.refVacuumProccess.xStopUnit:=FALSE;
		THIS^.StopUnitProcessStage:=StopUnitStage.CLOSE_BAV3_BIG;
	StopUnitStage.CLOSE_BAV3_BIG:
		THIS^.refBAV3Big.xAutoCommand:=FALSE;
		IF THIS^.refBAV3Big.xClosed THEN
			THIS^.StopUnitProcessStage:=StopUnitStage.CLOSE_BAV3_SMALL;
		END_IF
	StopUnitStage.CLOSE_BAV3_SMALL:
		THIS^.refBAV3Small.xAutoCommand:=FALSE;
		IF THIS^.refBAV3Small.xClosed THEN
			THIS^.StopUnitProcessStage:=StopUnitStage.CLOSE_BAV1_BIG;
		END_IF
	StopUnitStage.CLOSE_BAV1_BIG:
		THIS^.refBAV1Big.xAutoCommand:=FALSE;
		IF THIS^.refBAV1Big.xClosed THEN
			THIS^.StopUnitProcessStage:=StopUnitStage.CLOSE_BAV1_SMALL;
		END_IF
	StopUnitStage.CLOSE_BAV1_SMALL:
		THIS^.refBAV1Small.xAutoCommand:=FALSE;
		IF THIS^.refBAV1Small.xClosed THEN
			THIS^.StopUnitProcessStage:=StopUnitStage.TURNOFF_TMP;
		END_IF
	StopUnitStage.TURNOFF_TMP:
		THIS^.refTMP.xAutoCommand:=FALSE;
		IF THIS^.refTMP.xPumpNotOperating THEN
			THIS^.StopUnitProcessStage:=StopUnitStage.CLOSE_BAV2;
		END_IF
	StopUnitStage.CLOSE_BAV2:
		THIS^.refBAV2.xAutoCommand:=FALSE;
		IF THIS^.refBAV2.xClosed THEN
			THIS^.StopUnitProcessStage:=StopUnitStage.TURNOFF_FVP;
		END_IF
	StopUnitStage.TURNOFF_FVP:
		THIS^.refFVP.xAutoCommand:=FALSE;
		IF NOT THIS^.refFVP.xTurnOn THEN
			THIS^.StopUnitProcessStage:=StopUnitStage.COMPLETE;
		END_IF
	StopUnitStage.COMPLETE:
		THIS^.StopUnitProcessStage:=StopUnitStage.WAIT;
		THIS^.StopUnitProcessComplete:=TRUE;
	StopUnitStage.ERROR:
		THIS^.StopUnitProcessError:=TRUE;
	
END_CASE
END_METHOD

METHOD PRIVATE ValveOpen
VAR_INPUT
	Valve: REFERENCE TO udtValve;
	Stage: REFERENCE TO INT;
	Pressure: REFERENCE TO REAL;
	ErrorStage:INT;
	NextStage: INT;
END_VAR
		IF Valve.xClosed THEN
			Valve.xAutoCommand:=TRUE;
		END_IF	
		IF Valve.xError THEN
			Valve.xAutoCommand:=FALSE;
			Stage:=ErrorStage;
		END_IF
		IF Valve.xOpened AND (THIS^.refCameraPressure.rPressure <= Pressure) THEN
			Stage:=NextStage;
		END_IF
END_METHOD

METHOD PROTECTED _commandHandler : WORD
VAR_INPUT
END_VAR
VAR
	_wResetProcessStatus: WORD;
END_VAR
_wResetProcessStatus:=THIS^._resetProcess();
IF _wResetProcessStatus = 200 THEN
	RETURN;
END_IF
IF THIS^._xCommandLock THEN
	THIS^._resetAllCommand();
ELSE
	THIS^._commandRouter();	
END_IF
END_METHOD

//Выбло стадии в зависимости от комманды пользователя
METHOD PROTECTED _commandRouter : WORD
VAR_INPUT
END_VAR
IF THIS^.refVacuumProccess.xStartUnit THEN
	THIS^._xCommandLock:=TRUE;
	THIS^._iNextStage:=VacuumStage.START_UNIT;
	RETURN;
END_IF
IF THIS^.refVacuumProccess.xStopUnit THEN
	THIS^._xCommandLock:=TRUE;
	THIS^._iNextStage:=VacuumStage.STOP_UNIT;
END_IF
IF THIS^.refVacuumProccess.xStartDevacuumProcess THEN
	THIS^._xCommandLock:=TRUE;
	THIS^._iNextStage:=VacuumStage.DEVACUUM;
END_IF
IF THIS^.refVacuumProccess.xStartRevacuumProccess THEN
	THIS^._xCommandLock:=TRUE;
	THIS^._iNextStage:=VacuumStage.REVACUUM;
END_IF
END_METHOD

METHOD PROTECTED _resetAllCommand : WORD
VAR_INPUT
END_VAR
	THIS^.refVacuumProccess.xStartDevacuumProcess:=FALSE;
	THIS^.refVacuumProccess.xStartUnit:=FALSE;
	THIS^.refVacuumProccess.xStartDevacuumProcess:=FALSE;
	THIS^.refVacuumProccess.xStartRevacuumProccess:=FALSE;
END_METHOD

METHOD PROTECTED _resetProcess : WORD
VAR_INPUT
END_VAR
IF THIS^.refVacuumProccess.xResetProcess THEN
	THIS^.refVacuumProccess.xResetProcess := FALSE;
	THIS^._iNextStage:=VacuumStage.RESET_PROCESS;
	_resetProcess:=200;
ELSE
	_resetProcess:=0;
END_IF
END_METHOD

PROPERTY PUBLIC isAllvalveClosed : BOOL
GET
isAllvalveClosed:=THIS^.refBAV1Big.xClosed AND THIS^.refBAV1Small.xClosed AND THIS^.refBAV2.xClosed AND THIS^.refBAV3Big.xClosed AND THIS^.refBAV3Small.xClosed AND THIS^.refSHV.xClosed;
END_GET
END_PROPERTY

END_FUNCTION_BLOCK

// Function Blocks/VacuumSensore/ConverExp/ConverPressureToHmi
FUNCTION ConverPressureToHmi : BOOL
VAR_INPUT
	SourcePressure: REAL;
	ExpPressure: REFERENCE TO ExpPressure;
END_VAR
VAR
END_VAR

IF SourcePressure > 1.0 THEN
	More(Pressure:=SourcePressure,
		 ExpPressure:=ExpPressure);
ELSIF SourcePressure > 0.0 AND SourcePressure <= 1.0 THEN
	LessPressure(Pressure2:=SourcePressure,
		 HMIPressure2:=ExpPressure);
END_IF

END_FUNCTION

// Function Blocks/VacuumSensore/ConverExp/More
FUNCTION More : BOOL
VAR_INPUT
	Pressure: REAL;
	ExpPressure: REFERENCE TO ExpPressure;
END_VAR
VAR
	k:INT:=0;
	data:REAL:=0.0;
END_VAR

data:=Pressure;
WHILE data >10 DO
	k:=k+1;
	data:=data/10;
END_WHILE
ExpPressure.Exponenta:=k;
ExpPressure.Mantisa.rPressure:=data;

END_FUNCTION

// Function Blocks/VacuumSensore/ConverExp/LessPressure
FUNCTION LessPressure : BOOL
VAR_INPUT
	Pressure2: REAL;
	HMIPressure2: REFERENCE TO ExpPressure;
END_VAR
VAR
	k:INT:=0;
	data:REAL:=0.0;
END_VAR

data:=Pressure2;
WHILE data <= 1.0 DO
	k:=k-1;
	data:=data*10;
END_WHILE
HMIPressure2.Exponenta:=k;
HMIPressure2.Mantisa.rPressure:=data;

END_FUNCTION
